# EPICS substitutions: dependancyFiles/motorSim_motor.substitutions
file "$(MOTOR)/db/basic_asyn_motor.db"
{
pattern
{P,     N,  M,        DTYP,         PORT,       ADDR,  DESC,          EGU,      DIR,  VELO,  VBAS,  ACCL,  BDST,  BVEL,  BACC,  MRES,  PREC,  DHLM,  DLLM,  INIT}
{$(PREFIX),  1,  "m$(N)",  "asynMotor",  motorSim1,  0,     "motor $(N)",  degrees,  Pos,  1,     .1,    .2,    0,     1,     .2,    0.01,  5,     100,   -100,  ""}
{$(PREFIX),  2,  "m$(N)",  "asynMotor",  motorSim1,  1,     "motor $(N)",  degrees,  Pos,  1,     .1,    .2,    0,     1,     .2,    0.01,  5,     100,   -100,  ""}
{$(PREFIX),  3,  "m$(N)",  "asynMotor",  motorSim1,  2,     "motor $(N)",  degrees,  Pos,  1,     .1,    .2,    0,     1,     .2,    0.01,  5,     100,   -100,  ""}
{$(PREFIX),  4,  "m$(N)",  "asynMotor",  motorSim1,  3,     "motor $(N)",  degrees,  Pos,  1,     .1,    .2,    0,     1,     .2,    0.01,  5,     100,   -100,  ""}

{$(PREFIX),  5,  "m$(N)",  "asynMotor",  motorSim2,  0,     "motor $(N)",  degrees,  Pos,  1,     .1,    .2,    0,     1,     .2,    0.01,  5,     100,   -100,  ""}
{$(PREFIX),  6,  "m$(N)",  "asynMotor",  motorSim2,  1,     "motor $(N)",  degrees,  Pos,  1,     .1,    .2,    0,     1,     .2,    0.01,  5,     100,   -100,  ""}
{$(PREFIX),  7,  "m$(N)",  "asynMotor",  motorSim2,  2,     "motor $(N)",  degrees,  Pos,  1,     .1,    .2,    0,     1,     .2,    0.01,  5,     100,   -100,  ""}
{$(PREFIX),  8,  "m$(N)",  "asynMotor",  motorSim2,  3,     "motor $(N)",  degrees,  Pos,  1,     .1,    .2,    0,     1,     .2,    0.01,  5,     100,   -100,  ""}
}
